FUNCTION_BLOCK Recipe_10018_TripleCookiemitTopping
VAR_INPUT
	execute	: BOOL;
	Order	: DUT_RECIPEORDER;
END_VAR
VAR_OUTPUT
	RecipeInfo	: DUT_RECIPEOFFER;
	RecipeDone	: BOOL;	
	InitDone	: BOOL;
END_VAR
VAR
	StepDone	: BOOL;
	Layercnt	: INT := 0;
	OrderLayers	: INT := 2;
	i : INT;
END_VAR

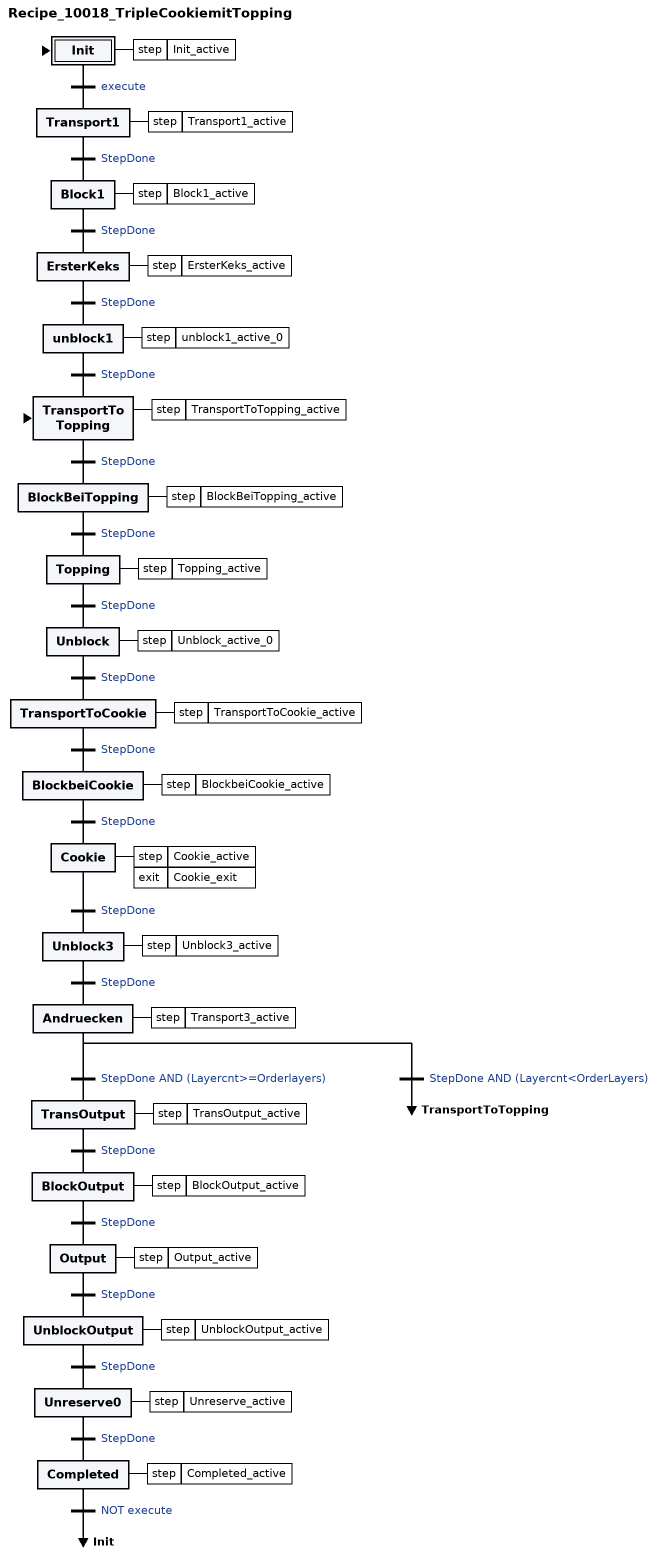
INITIAL_STEP Init:
    Init_active(N);  // step action
END_STEP
TRANSITION FROM Init TO Transport1
    := execute;
END_TRANSITION
STEP Transport1:
    Transport1_active(N);  // step action
END_STEP
TRANSITION FROM Transport1 TO Block1
    := StepDone;
END_TRANSITION
STEP Block1:
    Block1_active(N);  // step action
END_STEP
TRANSITION FROM Block1 TO ErsterKeks
    := StepDone;
END_TRANSITION
STEP ErsterKeks:
    ErsterKeks_active(N);  // step action
END_STEP
TRANSITION FROM ErsterKeks TO unblock1
    := StepDone;
END_TRANSITION
STEP unblock1:
    unblock1_active_0(N);  // step action
END_STEP
TRANSITION FROM unblock1 TO TransportToTopping
    := StepDone;
END_TRANSITION
STEP TransportToTopping:
    TransportToTopping_active(N);  // step action
END_STEP
TRANSITION FROM TransportToTopping TO BlockBeiTopping
    := StepDone;
END_TRANSITION
STEP BlockBeiTopping:
    BlockBeiTopping_active(N);  // step action
END_STEP
TRANSITION FROM BlockBeiTopping TO Topping
    := StepDone;
END_TRANSITION
STEP Topping:
    Topping_active(N);  // step action
END_STEP
TRANSITION FROM Topping TO Unblock
    := StepDone;
END_TRANSITION
STEP Unblock:
    Unblock_active_0(N);  // step action
END_STEP
TRANSITION FROM Unblock TO TransportToCookie
    := StepDone;
END_TRANSITION
STEP TransportToCookie:
    TransportToCookie_active(N);  // step action
END_STEP
TRANSITION FROM TransportToCookie TO BlockbeiCookie
    := StepDone;
END_TRANSITION
STEP BlockbeiCookie:
    BlockbeiCookie_active(N);  // step action
END_STEP
TRANSITION FROM BlockbeiCookie TO Cookie
    := StepDone;
END_TRANSITION
STEP Cookie:
    Cookie_active(N);  // step action
    Cookie_exit(P0);  // exit action
END_STEP
TRANSITION FROM Cookie TO Unblock3
    := StepDone;
END_TRANSITION
STEP Unblock3:
    Unblock3_active(N);  // step action
END_STEP
TRANSITION FROM Unblock3 TO Andruecken
    := StepDone;
END_TRANSITION
STEP Andruecken:
    Transport3_active(N);  // step action
END_STEP
TRANSITION FROM Andruecken TO TransOutput
    := StepDone AND (Layercnt>=Orderlayers);
END_TRANSITION
STEP TransOutput:
    TransOutput_active(N);  // step action
END_STEP
TRANSITION FROM TransOutput TO BlockOutput
    := StepDone;
END_TRANSITION
STEP BlockOutput:
    BlockOutput_active(N);  // step action
END_STEP
TRANSITION FROM BlockOutput TO Output
    := StepDone;
END_TRANSITION
STEP Output:
    Output_active(N);  // step action
END_STEP
TRANSITION FROM Output TO UnblockOutput
    := StepDone;
END_TRANSITION
STEP UnblockOutput:
    UnblockOutput_active(N);  // step action
END_STEP
TRANSITION FROM UnblockOutput TO Unreserve0
    := StepDone;
END_TRANSITION
TRANSITION FROM Andruecken TO TransportToTopping
    := StepDone AND (Layercnt<OrderLayers);
END_TRANSITION
STEP Unreserve0:
    Unreserve_active(N);  // step action
END_STEP
TRANSITION FROM Unreserve0 TO Completed
    := StepDone;
END_TRANSITION
STEP Completed:
    Completed_active(N);  // step action
END_STEP
TRANSITION FROM Completed TO Init
    := NOT execute;
END_TRANSITION

ACTION BlockOutput_active:
StepDone := FALSE;

//Skill auswählen



ExecuteSkill.SkillID 		:= 1315;
ExecuteSkill.SkillName	 	:= 'Block';

ExecuteSkill();

StepDone := ExecuteSkill.Done;
END_ACTION

ACTION Production2_active:
StepDone := FALSE;
RecipeDone := FALSE;
//Skill auswählen
ExecuteSkill.SkillID 		:= 1339;
ExecuteSkill.SkillName	 	:= 'ParameterTESTSKILL1339';


ExecuteSkill.Parameter[0].ID := 10;
ExecuteSkill.Parameter[0].Name := 'Blinkfrequenz';
ExecuteSkill.Parameter[0].Value := Order.UserParameter[0].Value*2;


ExecuteSkill();

StepDone := ExecuteSkill.Done;
END_ACTION

ACTION TransportToCookie_active:
StepDone := FALSE;

//Skill auswählen
ExecuteSkill.SkillID 		:= 1320;
ExecuteSkill.SkillName	 	:= 'Transport';

//Parameter setzen

ExecuteSkill.Parameter[3].ID := 3;
ExecuteSkill.Parameter[3].Name := 'Velocity';
ExecuteSkill.Parameter[3].Value := 400;



ExecuteSkill.Parameter[1].ID :=  1;
ExecuteSkill.Parameter[1].Name := 'TargetPosition X';
ExecuteSkill.Parameter[1].Value := 30 ;
ExecuteSkill.Parameter[1].StringValue := '#DP#2#XPosition';



ExecuteSkill.Parameter[2].ID := 2;
ExecuteSkill.Parameter[2].Name := 'TargetPosition Z';
ExecuteSkill.Parameter[2].Value := ZCookieModule + ZCookieModuleCalibration - ((Layercnt +1) * ( toppingthickness - cookiethickness)) ;

ExecuteSkill();

StepDone := ExecuteSkill.Done;
END_ACTION

ACTION Topping_active:
StepDone := FALSE;

//Skill auswählen
CASE REAL_TO_INT (order.UserParameter[2*LayerCnt].Value) OF
	1: 
		ExecuteSkill.SkillID 		:=  1230;
		ExecuteSkill.SkillName	 	:= 'Strawberry Topping';
	2: 
		ExecuteSkill.SkillID 		:=  1240;
		ExecuteSkill.SkillName	 	:= 'Apple Topping';
	ELSE
		ExecuteSkill.SkillID 		:=  1230;
		ExecuteSkill.SkillName	 	:= 'Strawberry Topping';
END_CASE


//Parameter setzen

ExecuteSkill.Parameter[0].ID := 1;
ExecuteSkill.Parameter[0].Name := 'Amount';
ExecuteSkill.Parameter[0].Value := order.UserParameter[2*LayerCnt + 1].Value ;


(*
ExecuteSkill.Parameter[1].ID := 1;
ExecuteSkill.Parameter[1].Name := 'TaskID';
ExecuteSkill.Parameter[1].Value := 130;
*)
(*
ExecuteSkill.Parameter[2].ID := ;
ExecuteSkill.Parameter[2].Name := '';
ExecuteSkill.Parameter[2].Value := ;
*)

(*
ExecuteSkill.Parameter[3].ID := ;
ExecuteSkill.Parameter[3].Name := '';
ExecuteSkill.Parameter[3].Value := ;
*)

(*
ExecuteSkill.Parameter[4].ID := ;
ExecuteSkill.Parameter[4].Name := '';
ExecuteSkill.Parameter[4].Value := ;
*)

(*
ExecuteSkill.Parameter[5].ID := ;
ExecuteSkill.Parameter[5].Name := '';
ExecuteSkill.Parameter[5].Value := ;
*)

ExecuteSkill();

StepDone := ExecuteSkill.Done;
END_ACTION

ACTION BlockbeiCookie_active:
StepDone := FALSE;

//Skill auswählen
ExecuteSkill.SkillID 		:= 1315;
ExecuteSkill.SkillName	 	:= 'Block';

//Parameter setzen

ExecuteSkill.Parameter[1].ID := 1;
ExecuteSkill.Parameter[1].Name := 'TaskID';
ExecuteSkill.Parameter[1].Value := 130;


(*
ExecuteSkill.Parameter[2].ID := ;
ExecuteSkill.Parameter[2].Name := '';
ExecuteSkill.Parameter[2].Value := ;
*)

(*
ExecuteSkill.Parameter[3].ID := ;
ExecuteSkill.Parameter[3].Name := '';
ExecuteSkill.Parameter[3].Value := ;
*)

(*
ExecuteSkill.Parameter[4].ID := ;
ExecuteSkill.Parameter[4].Name := '';
ExecuteSkill.Parameter[4].Value := ;
*)

(*
ExecuteSkill.Parameter[5].ID := ;
ExecuteSkill.Parameter[5].Name := '';
ExecuteSkill.Parameter[5].Value := ;
*)



ExecuteSkill();

StepDone := ExecuteSkill.Done;
END_ACTION

ACTION Unblock1_active:
StepDone := FALSE;

//Skill auswählen

CASE LREAL_TO_INT (order.UserParameter[2].Value) OF

1:
ExecuteSkill.SkillID 		:= 1316;
ExecuteSkill.SkillName	 	:= 'Unblock';

ExecuteSkill();

StepDone := ExecuteSkill.Done;
ELSE StepDone := TRUE;

END_CASE
END_ACTION

ACTION Transport_active:
StepDone := FALSE;

//Skill auswählen

CASE LREAL_TO_INT (order.UserParameter[2].Value) OF

1:
//Skill auswählen
ExecuteSkill.SkillID 		:= 1320;
ExecuteSkill.SkillName	 	:= 'Transport';

//Parameter setzen

ExecuteSkill.Parameter[3].ID :=3 ;
ExecuteSkill.Parameter[3].Name := 'Velocity';
ExecuteSkill.Parameter[3].Value := 1500;



ExecuteSkill.Parameter[1].ID :=1 ;
ExecuteSkill.Parameter[1].Name := 'TargetPosition X';
ExecuteSkill.Parameter[1].StringValue := '#DP#2#XPosition';
ExecuteSkill.Parameter[1].Value := 200 ;


ExecuteSkill.Parameter[2].ID := 2 ;
ExecuteSkill.Parameter[2].Name := 'TargetPosition Z';
ExecuteSkill.Parameter[2].Value := 90 ;



ExecuteSkill.Parameter[4].ID := 4 ;
ExecuteSkill.Parameter[4].Name := 'Acceleration';
ExecuteSkill.Parameter[4].Value := 4500;


(*
ExecuteSkill.Parameter[5].ID := ;
ExecuteSkill.Parameter[5].Name := '';
ExecuteSkill.Parameter[5].Value := ;
*)



ExecuteSkill();

StepDone := ExecuteSkill.Done;
ELSE StepDone := TRUE;

END_CASE
END_ACTION

ACTION Transport2_active:
StepDone := FALSE;

//Skill auswählen
ExecuteSkill.SkillID 		:= 1320;
ExecuteSkill.SkillName	 	:= 'Transport';

//Parameter setzen

ExecuteSkill.Parameter[3].ID := 3;
ExecuteSkill.Parameter[3].Name := 'Velocity';
ExecuteSkill.Parameter[3].Value := 2800;



ExecuteSkill.Parameter[1].ID :=  1;
ExecuteSkill.Parameter[1].Name := 'TargetPosition X';
ExecuteSkill.Parameter[1].Value := 30 ;
ExecuteSkill.Parameter[1].StringValue := '#DP#2#XPosition';



ExecuteSkill.Parameter[2].ID := 2;
ExecuteSkill.Parameter[2].Name := 'TargetPosition Z';
ExecuteSkill.Parameter[2].Value := 0 ;



ExecuteSkill.Parameter[4].ID := 4;
ExecuteSkill.Parameter[4].Name := 'Acceleration';
ExecuteSkill.Parameter[4].Value := 2000 ;


(*
ExecuteSkill.Parameter[5].ID := ;
ExecuteSkill.Parameter[5].Name := '';
ExecuteSkill.Parameter[5].Value := ;
*)



ExecuteSkill();

StepDone := ExecuteSkill.Done;
END_ACTION

ACTION Block2_active:
StepDone := FALSE;

//Skill auswählen
ExecuteSkill.SkillID 		:= 1315;
ExecuteSkill.SkillName	 	:= 'Block';

//Parameter setzen

ExecuteSkill.Parameter[1].ID := 1;
ExecuteSkill.Parameter[1].Name := 'TaskID';
ExecuteSkill.Parameter[1].Value := 130;


(*
ExecuteSkill.Parameter[2].ID := ;
ExecuteSkill.Parameter[2].Name := '';
ExecuteSkill.Parameter[2].Value := ;
*)

(*
ExecuteSkill.Parameter[3].ID := ;
ExecuteSkill.Parameter[3].Name := '';
ExecuteSkill.Parameter[3].Value := ;
*)

(*
ExecuteSkill.Parameter[4].ID := ;
ExecuteSkill.Parameter[4].Name := '';
ExecuteSkill.Parameter[4].Value := ;
*)

(*
ExecuteSkill.Parameter[5].ID := ;
ExecuteSkill.Parameter[5].Name := '';
ExecuteSkill.Parameter[5].Value := ;
*)



ExecuteSkill();

StepDone := ExecuteSkill.Done;
END_ACTION

ACTION Reserve_active:
StepDone := FALSE;
RecipeDone := FALSE;
//Skill auswählen
ExecuteSkill.SkillID 		:= 1310;
ExecuteSkill.SkillName	 	:= 'Reserve';

//Parameter setzen

ExecuteSkill.Parameter[1].ID := 1;
ExecuteSkill.Parameter[1].Name := 'TaskID';
ExecuteSkill.Parameter[1].Value := 123;


(*
ExecuteSkill.Parameter[2].ID := ;
ExecuteSkill.Parameter[2].Name := '';
ExecuteSkill.Parameter[2].Value := ;
*)

(*
ExecuteSkill.Parameter[3].ID := ;
ExecuteSkill.Parameter[3].Name := '';
ExecuteSkill.Parameter[3].Value := ;
*)

(*
ExecuteSkill.Parameter[4].ID := ;
ExecuteSkill.Parameter[4].Name := '';
ExecuteSkill.Parameter[4].Value := ;
*)

(*
ExecuteSkill.Parameter[5].ID := ;
ExecuteSkill.Parameter[5].Name := '';
ExecuteSkill.Parameter[5].Value := ;
*)



ExecuteSkill();

StepDone := ExecuteSkill.Done;
END_ACTION

ACTION Unblock_active:
StepDone := FALSE;

//Skill auswählen
ExecuteSkill.SkillID 		:= 1316;
ExecuteSkill.SkillName	 	:= 'Unblock';

//Parameter setzen

ExecuteSkill.Parameter[1].ID := 1;
ExecuteSkill.Parameter[1].Name := 'TaskID';
ExecuteSkill.Parameter[1].Value := 125;


(*
ExecuteSkill.Parameter[2].ID := ;
ExecuteSkill.Parameter[2].Name := '';
ExecuteSkill.Parameter[2].Value := ;
*)

(*
ExecuteSkill.Parameter[3].ID := ;
ExecuteSkill.Parameter[3].Name := '';
ExecuteSkill.Parameter[3].Value := ;
*)

(*
ExecuteSkill.Parameter[4].ID := ;
ExecuteSkill.Parameter[4].Name := '';
ExecuteSkill.Parameter[4].Value := ;
*)

(*
ExecuteSkill.Parameter[5].ID := ;
ExecuteSkill.Parameter[5].Name := '';
ExecuteSkill.Parameter[5].Value := ;
*)



ExecuteSkill();

StepDone := ExecuteSkill.Done;
END_ACTION

ACTION Cookie_active:
StepDone := FALSE;
RecipeDone := FALSE;
//Skill auswählen
ExecuteSkill.SkillID 		:= 1010;
ExecuteSkill.SkillName	 	:= 'Cookie ausgeben';





ExecuteSkill();

StepDone := ExecuteSkill.Done;
END_ACTION

ACTION TransOutput_active:
StepDone := FALSE;

//Skill auswählen
ExecuteSkill.SkillID 		:= 1320;
ExecuteSkill.SkillName	 	:= 'Name';

//Parameter setzen

ExecuteSkill.Parameter[3].ID := 3;
ExecuteSkill.Parameter[3].Name := 'Velocity';
ExecuteSkill.Parameter[3].Value := 1500;



ExecuteSkill.Parameter[4].ID := 4 ;
ExecuteSkill.Parameter[4].Name := 'Acceleration';
ExecuteSkill.Parameter[4].Value := 1000 ;



ExecuteSkill.Parameter[1].ID := 1;
ExecuteSkill.Parameter[1].Name := 'TargetPosition X';
ExecuteSkill.Parameter[1].Value := 3200 ;
ExecuteSkill.Parameter[1].StringValue := '#DP#2#XPosition' ;




ExecuteSkill.Parameter[2].ID := 2;
ExecuteSkill.Parameter[2].Name := 'TargetPosition Z';
ExecuteSkill.Parameter[2].Value := ZInputOutput;


(*
ExecuteSkill.Parameter[5].ID := ;
ExecuteSkill.Parameter[5].Name := '';
ExecuteSkill.Parameter[5].Value := ;
*)



ExecuteSkill();

StepDone := ExecuteSkill.Done;
END_ACTION

ACTION TransportToTopping_active:
StepDone := FALSE;

//Skill auswählen
ExecuteSkill.SkillID 		:= 1320;
ExecuteSkill.SkillName	 	:= 'Transport';

//Parameter setzen

ExecuteSkill.Parameter[3].ID := 3;
ExecuteSkill.Parameter[3].Name := 'Velocity';
ExecuteSkill.Parameter[3].Value := 1000;



ExecuteSkill.Parameter[1].ID :=  1;
ExecuteSkill.Parameter[1].Name := 'TargetPosition X';
ExecuteSkill.Parameter[1].Value := 30 ;
ExecuteSkill.Parameter[1].StringValue := '#DP#2#XPosition';



ExecuteSkill.Parameter[2].ID := 2;
ExecuteSkill.Parameter[2].Name := 'TargetPosition Z';
ExecuteSkill.Parameter[2].Value := ZCremeModule + ZCremeModuleCalibration - Layercnt * ( cookiethickness + toppingthickness);

ExecuteSkill();

StepDone := ExecuteSkill.Done;
END_ACTION

ACTION Unblock_active_0:
StepDone := FALSE;

//Skill auswählen
ExecuteSkill.SkillID 		:= 1316;
ExecuteSkill.SkillName	 	:= 'Unblock';

//Parameter setzen

ExecuteSkill.Parameter[1].ID := 1;
ExecuteSkill.Parameter[1].Name := 'TaskID';
ExecuteSkill.Parameter[1].Value := 128 ;


(*
ExecuteSkill.Parameter[2].ID := ;
ExecuteSkill.Parameter[2].Name := '';
ExecuteSkill.Parameter[2].Value := ;
*)

(*
ExecuteSkill.Parameter[3].ID := ;
ExecuteSkill.Parameter[3].Name := '';
ExecuteSkill.Parameter[3].Value := ;
*)

(*
ExecuteSkill.Parameter[4].ID := ;
ExecuteSkill.Parameter[4].Name := '';
ExecuteSkill.Parameter[4].Value := ;
*)

(*
ExecuteSkill.Parameter[5].ID := ;
ExecuteSkill.Parameter[5].Name := '';
ExecuteSkill.Parameter[5].Value := ;
*)



ExecuteSkill();

StepDone := ExecuteSkill.Done;
END_ACTION

ACTION Cookie_exit:
Layercnt := Layercnt +1;
END_ACTION

ACTION Block0_active:
StepDone := FALSE;

//Skill auswählen

CASE LREAL_TO_INT (order.UserParameter[2].Value) OF

1:
ExecuteSkill.SkillID 		:= 1315;
ExecuteSkill.SkillName	 	:= 'Block';

ExecuteSkill();

StepDone := ExecuteSkill.Done;
ELSE StepDone := TRUE;

END_CASE
END_ACTION

ACTION BlockBeiTopping_active:
StepDone := FALSE;

//Skill auswählen
ExecuteSkill.SkillID 		:= 1315;
ExecuteSkill.SkillName	 	:= 'Block';

//Parameter setzen

ExecuteSkill.Parameter[1].ID := 1;
ExecuteSkill.Parameter[1].Name := 'TaskID';
ExecuteSkill.Parameter[1].Value := 130;


(*
ExecuteSkill.Parameter[2].ID := ;
ExecuteSkill.Parameter[2].Name := '';
ExecuteSkill.Parameter[2].Value := ;
*)

(*
ExecuteSkill.Parameter[3].ID := ;
ExecuteSkill.Parameter[3].Name := '';
ExecuteSkill.Parameter[3].Value := ;
*)

(*
ExecuteSkill.Parameter[4].ID := ;
ExecuteSkill.Parameter[4].Name := '';
ExecuteSkill.Parameter[4].Value := ;
*)

(*
ExecuteSkill.Parameter[5].ID := ;
ExecuteSkill.Parameter[5].Name := '';
ExecuteSkill.Parameter[5].Value := ;
*)



ExecuteSkill();

StepDone := ExecuteSkill.Done;
END_ACTION

ACTION Completed_active:
RecipeDone := TRUE;
StepDone := FALSE;
Layercnt := 0;
END_ACTION

ACTION ErsterKeks_active:
StepDone := FALSE;
RecipeDone := FALSE;
//Skill auswählen
ExecuteSkill.SkillID 		:= 1010;
ExecuteSkill.SkillName	 	:= 'Seperate Cookie';


ExecuteSkill();

StepDone := ExecuteSkill.Done;
END_ACTION

ACTION Output_active:
StepDone := FALSE;

//Skill auswählen
ExecuteSkill.SkillID 		:= 1403;
ExecuteSkill.SkillName	 	:= 'Output';

//Parameter setzen

ExecuteSkill.Parameter[1].ID := 1;
ExecuteSkill.Parameter[1].Name := 'TaskID';
ExecuteSkill.Parameter[1].Value := Order.TaskID;


(*
ExecuteSkill.Parameter[2].ID := ;
ExecuteSkill.Parameter[2].Name := '';
ExecuteSkill.Parameter[2].Value := ;
*)

(*
ExecuteSkill.Parameter[3].ID := ;
ExecuteSkill.Parameter[3].Name := '';
ExecuteSkill.Parameter[3].Value := ;
*)

(*
ExecuteSkill.Parameter[4].ID := ;
ExecuteSkill.Parameter[4].Name := '';
ExecuteSkill.Parameter[4].Value := ;
*)

(*
ExecuteSkill.Parameter[5].ID := ;
ExecuteSkill.Parameter[5].Name := '';
ExecuteSkill.Parameter[5].Value := ;
*)



ExecuteSkill();

StepDone := ExecuteSkill.Done;
END_ACTION

ACTION Block1_active:
StepDone := FALSE;

//Skill auswählen
ExecuteSkill.SkillID 		:= 1315;
ExecuteSkill.SkillName	 	:= 'Block';

//Parameter setzen

ExecuteSkill.Parameter[1].ID := 1;
ExecuteSkill.Parameter[1].Name := 'TaskID';
ExecuteSkill.Parameter[1].Value := 127;


(*
ExecuteSkill.Parameter[2].ID := ;
ExecuteSkill.Parameter[2].Name := '';
ExecuteSkill.Parameter[2].Value := ;
*)

(*
ExecuteSkill.Parameter[3].ID := ;
ExecuteSkill.Parameter[3].Name := '';
ExecuteSkill.Parameter[3].Value := ;
*)

(*
ExecuteSkill.Parameter[4].ID := ;
ExecuteSkill.Parameter[4].Name := '';
ExecuteSkill.Parameter[4].Value := ;
*)

(*
ExecuteSkill.Parameter[5].ID := ;
ExecuteSkill.Parameter[5].Name := '';
ExecuteSkill.Parameter[5].Value := ;
*)



ExecuteSkill();

StepDone := ExecuteSkill.Done;
END_ACTION

ACTION Init_active:
RecipeDone := FALSE;

// Initialisation of Recipe Parameters an name etc
RecipeInfo.Name := 'Triple Cookie';
RecipeInfo.Description := 'Three Butter Cookies framing your choosen Toppings';
RecipeInfo.Dummy := FALSE;
RecipeInfo.RecipeID := 10018;	// 
Initdone := TRUE;
FOR i := 0 TO UserParameterCnt DO
	IF Order.UserParameter[i].Value = 0 THEN
		order.UserParameter[i].Value := RecipeInfo.UserParameter[i].Default;
	END_IF
END_FOR

//Parameter 0:

	RecipeInfo.UserParameter[0].Dummy 		:= FALSE;
	RecipeInfo.UserParameter[0].Default		:= 1;
	RecipeInfo.UserParameter[0].Description	:= 'Choose your first Topping (Top Layer)';
	RecipeInfo.UserParameter[0].MaxValue	:= 2;
	RecipeInfo.UserParameter[0].MinValue	:= 1;
	RecipeInfo.UserParameter[0].Name		:= 'Topping';
	RecipeInfo.UserParameter[0].Unit		:= 'Strawberry, Apple';
	RecipeInfo.UserParameter[0].Step		:= 1;

//Parameter 1:

	RecipeInfo.UserParameter[1].Dummy 		:= FALSE;
	RecipeInfo.UserParameter[1].Default		:= 50;
	RecipeInfo.UserParameter[1].Description	:= 'Amount of the selected Topping';
	RecipeInfo.UserParameter[1].MaxValue	:= 100;
	RecipeInfo.UserParameter[1].MinValue	:= 0;
	RecipeInfo.UserParameter[1].Name		:= 'Amount';
	RecipeInfo.UserParameter[1].Unit		:= '';
	RecipeInfo.UserParameter[1].Step		:= 1;

//Parameter 2:
	RecipeInfo.UserParameter[2].Dummy 		:= FALSE;
	RecipeInfo.UserParameter[2].Default		:= 2;
	RecipeInfo.UserParameter[2].Description	:= 'Choose weather you want to include a simulated module';
	RecipeInfo.UserParameter[2].MaxValue	:= 2;
	RecipeInfo.UserParameter[2].MinValue	:= 1;
	RecipeInfo.UserParameter[2].Name		:= 'Virtual Module';
	RecipeInfo.UserParameter[2].Unit		:= 'enabled, disabled';
	RecipeInfo.UserParameter[2].Step		:= 1;

//Parameter 3:
	RecipeInfo.UserParameter[3].Dummy 		:= FALSE;
	RecipeInfo.UserParameter[3].Default		:= 1;
	RecipeInfo.UserParameter[3].Description	:= 'Amount of the selected Topping';
	RecipeInfo.UserParameter[3].MaxValue	:= 100;
	RecipeInfo.UserParameter[3].MinValue	:= 0;
	RecipeInfo.UserParameter[3].Name		:= 'Amount';
	RecipeInfo.UserParameter[3].Unit		:= '';
	RecipeInfo.UserParameter[3].Step		:= 1;
//Parameter 4:

	RecipeInfo.UserParameter[4].Dummy 		:= FALSE;
	RecipeInfo.UserParameter[4].Default		:= 1;
	RecipeInfo.UserParameter[4].Description	:= 'Choose your third Topping';
	RecipeInfo.UserParameter[4].MaxValue	:= 2;
	RecipeInfo.UserParameter[4].MinValue	:= 1;
	RecipeInfo.UserParameter[4].Name		:= 'Topping';
	RecipeInfo.UserParameter[4].Unit		:= 'Strawberry, Apple';
	RecipeInfo.UserParameter[4].Step		:= 1;
	(*
//Parameter 5:

	RecipeInfo.UserParameter[5].Dummy 		:= FALSE;
	RecipeInfo.UserParameter[5].Default		:= 50;
	RecipeInfo.UserParameter[5].Description	:= 'Amount of the selected Topping';
	RecipeInfo.UserParameter[5].MaxValue	:= 100;
	RecipeInfo.UserParameter[5].MinValue	:= 0;
	RecipeInfo.UserParameter[5].Name		:= 'Amount';
	RecipeInfo.UserParameter[5].Unit		:= '';
	RecipeInfo.UserParameter[5].Step		:= 1;
*)
END_ACTION

ACTION Unblock3_active:
StepDone := FALSE;

//Skill auswählen
ExecuteSkill.SkillID 		:= 1316;
ExecuteSkill.SkillName	 	:= 'Unblock';

//Parameter setzen

ExecuteSkill.Parameter[1].ID := 1;
ExecuteSkill.Parameter[1].Name := 'TaskID';
ExecuteSkill.Parameter[1].Value := 131;


(*
ExecuteSkill.Parameter[2].ID := ;
ExecuteSkill.Parameter[2].Name := '';
ExecuteSkill.Parameter[2].Value := ;
*)

(*
ExecuteSkill.Parameter[3].ID := ;
ExecuteSkill.Parameter[3].Name := '';
ExecuteSkill.Parameter[3].Value := ;
*)

(*
ExecuteSkill.Parameter[4].ID := ;
ExecuteSkill.Parameter[4].Name := '';
ExecuteSkill.Parameter[4].Value := ;
*)

(*
ExecuteSkill.Parameter[5].ID := ;
ExecuteSkill.Parameter[5].Name := '';
ExecuteSkill.Parameter[5].Value := ;
*)



ExecuteSkill();

StepDone := ExecuteSkill.Done;
END_ACTION

ACTION Production0_active:
StepDone := FALSE;
RecipeDone := FALSE; 
//simulation ausgewählt?
CASE LREAL_TO_INT (order.UserParameter[2].Value) OF

1:
ExecuteSkill.SkillID 		:= 1337;
ExecuteSkill.SkillName	 	:= 'Testskill';

ExecuteSkill();

StepDone := ExecuteSkill.Done;
ELSE StepDone := TRUE;

END_CASE
END_ACTION

ACTION UnblockOutput_active:
StepDone := FALSE;

//Skill auswählen
ExecuteSkill.SkillID 		:= 1316;
ExecuteSkill.SkillName	 	:= 'Unblock';

//Parameter setzen



(*
ExecuteSkill.Parameter[2].ID := ;
ExecuteSkill.Parameter[2].Name := '';
ExecuteSkill.Parameter[2].Value := ;
*)

(*
ExecuteSkill.Parameter[3].ID := ;
ExecuteSkill.Parameter[3].Name := '';
ExecuteSkill.Parameter[3].Value := ;
*)

(*
ExecuteSkill.Parameter[4].ID := ;
ExecuteSkill.Parameter[4].Name := '';
ExecuteSkill.Parameter[4].Value := ;
*)

(*
ExecuteSkill.Parameter[5].ID := ;
ExecuteSkill.Parameter[5].Name := '';
ExecuteSkill.Parameter[5].Value := ;
*)



ExecuteSkill();

StepDone := ExecuteSkill.Done;
END_ACTION

ACTION Transport1_active:
StepDone := FALSE;

//Skill auswählen
ExecuteSkill.SkillID 		:= 1320;
ExecuteSkill.SkillName	 	:= 'Transport';

//Parameter setzen

ExecuteSkill.Parameter[3].ID := 3;
ExecuteSkill.Parameter[3].Name := 'Velocity';
ExecuteSkill.Parameter[3].Value := 1500;



ExecuteSkill.Parameter[4].ID := 4 ;
ExecuteSkill.Parameter[4].Name := 'Acceleration';
ExecuteSkill.Parameter[4].Value := 1000 ;



ExecuteSkill.Parameter[1].ID := 1;
ExecuteSkill.Parameter[1].Name := 'TargetPosition X';
ExecuteSkill.Parameter[1].Value := 3200 ;
ExecuteSkill.Parameter[1].StringValue := '#DP#2#XPosition' ;




ExecuteSkill.Parameter[2].ID := 2;
ExecuteSkill.Parameter[2].Name := 'TargetPosition Z';
ExecuteSkill.Parameter[2].Value := ZCookieModule + ZCocktailModuleCalibration;


(*
ExecuteSkill.Parameter[5].ID := ;
ExecuteSkill.Parameter[5].Name := '';
ExecuteSkill.Parameter[5].Value := ;
*)



ExecuteSkill();

StepDone := ExecuteSkill.Done;
END_ACTION

ACTION Unreserve_active:
StepDone := FALSE;

//Skill auswählen
ExecuteSkill.SkillID 		:= 1311;
ExecuteSkill.SkillName	 	:= 'Unreserve';

//Parameter setzen

ExecuteSkill.Parameter[1].ID := 1;
ExecuteSkill.Parameter[1].Name := 'TaskID';
ExecuteSkill.Parameter[1].Value := 131;


(*
ExecuteSkill.Parameter[2].ID := ;
ExecuteSkill.Parameter[2].Name := '';
ExecuteSkill.Parameter[2].Value := ;
*)

(*
ExecuteSkill.Parameter[3].ID := ;
ExecuteSkill.Parameter[3].Name := '';
ExecuteSkill.Parameter[3].Value := ;
*)

(*
ExecuteSkill.Parameter[4].ID := ;
ExecuteSkill.Parameter[4].Name := '';
ExecuteSkill.Parameter[4].Value := ;
*)

(*
ExecuteSkill.Parameter[5].ID := ;
ExecuteSkill.Parameter[5].Name := '';
ExecuteSkill.Parameter[5].Value := ;
*)



ExecuteSkill();

StepDone := ExecuteSkill.Done;
END_ACTION

ACTION Unblock2_active:
StepDone := FALSE;

//Skill auswählen
ExecuteSkill.SkillID 		:= 1316;
ExecuteSkill.SkillName	 	:= 'Unblock';

//Parameter setzen

ExecuteSkill.Parameter[1].ID := 1;
ExecuteSkill.Parameter[1].Name := 'TaskID';
ExecuteSkill.Parameter[1].Value := 131;


(*
ExecuteSkill.Parameter[2].ID := ;
ExecuteSkill.Parameter[2].Name := '';
ExecuteSkill.Parameter[2].Value := ;
*)

(*
ExecuteSkill.Parameter[3].ID := ;
ExecuteSkill.Parameter[3].Name := '';
ExecuteSkill.Parameter[3].Value := ;
*)

(*
ExecuteSkill.Parameter[4].ID := ;
ExecuteSkill.Parameter[4].Name := '';
ExecuteSkill.Parameter[4].Value := ;
*)

(*
ExecuteSkill.Parameter[5].ID := ;
ExecuteSkill.Parameter[5].Name := '';
ExecuteSkill.Parameter[5].Value := ;
*)



ExecuteSkill();

StepDone := ExecuteSkill.Done;
END_ACTION

ACTION unblock1_active_0:
StepDone := FALSE;

//Skill auswählen
ExecuteSkill.SkillID 		:= 1316;
ExecuteSkill.SkillName	 	:= 'Unblock';

//Parameter setzen

ExecuteSkill.Parameter[1].ID := 1;
ExecuteSkill.Parameter[1].Name := 'TaskID';
ExecuteSkill.Parameter[1].Value := 128 ;


(*
ExecuteSkill.Parameter[2].ID := ;
ExecuteSkill.Parameter[2].Name := '';
ExecuteSkill.Parameter[2].Value := ;
*)

(*
ExecuteSkill.Parameter[3].ID := ;
ExecuteSkill.Parameter[3].Name := '';
ExecuteSkill.Parameter[3].Value := ;
*)

(*
ExecuteSkill.Parameter[4].ID := ;
ExecuteSkill.Parameter[4].Name := '';
ExecuteSkill.Parameter[4].Value := ;
*)

(*
ExecuteSkill.Parameter[5].ID := ;
ExecuteSkill.Parameter[5].Name := '';
ExecuteSkill.Parameter[5].Value := ;
*)



ExecuteSkill();

StepDone := ExecuteSkill.Done;
END_ACTION

ACTION Transport3_active:
StepDone := FALSE;

//Skill auswählen
ExecuteSkill.SkillID 		:= 1320;
ExecuteSkill.SkillName	 	:= 'Transport';

//Parameter setzen

ExecuteSkill.Parameter[3].ID := 3;
ExecuteSkill.Parameter[3].Name := 'Velocity';
ExecuteSkill.Parameter[3].Value := 2800;



ExecuteSkill.Parameter[1].ID :=  1;
ExecuteSkill.Parameter[1].Name := 'TargetPosition X';
ExecuteSkill.Parameter[1].Value := 30 ;
ExecuteSkill.Parameter[1].StringValue := '#DP#-2#XPosition';



ExecuteSkill.Parameter[2].ID := 2;
ExecuteSkill.Parameter[2].Name := 'TargetPosition Z';
ExecuteSkill.Parameter[2].Value := 90;// ZCookieModule - ZCookieModuleCalibration - 2* Cookiethickness + toppingthickness+ Preasureheight  ;



ExecuteSkill.Parameter[4].ID := 4;
ExecuteSkill.Parameter[4].Name := 'Acceleration';
ExecuteSkill.Parameter[4].Value := 2000 ;


(*
ExecuteSkill.Parameter[5].ID := ;
ExecuteSkill.Parameter[5].Name := '';
ExecuteSkill.Parameter[5].Value := ;
*)



ExecuteSkill();

StepDone := ExecuteSkill.Done;
END_ACTION

END_FUNCTION_BLOCK

(* stored: Version 1.1.0.1, ProductVersion 3.1.0.25
   POU Recipe_10018_TripleCookiemitTopping: Id {35c293d9-a855-4621-991c-8fe2beba9ca6}
   Action BlockOutput_active: Id {074446d1-89b8-4d20-8427-d08b08451a01}
   Action Production2_active: Id {13fb47f7-1ed2-4213-80f0-7c79adf1d406}
   Action TransportToCookie_active: Id {17af7920-8f39-413e-ad0e-663d0bcc4454}
   Action Topping_active: Id {2cb82c9a-a023-458b-86f8-a51686875beb}
   Action BlockbeiCookie_active: Id {33ebe683-30f4-45d2-a737-c9de8ad1aa17}
   Action Unblock1_active: Id {3a205016-96c4-4631-8085-d6e13121b8ed}
   Action Transport_active: Id {50522275-ebaf-458e-95c2-2c4e8c56eb8e}
   Action Transport2_active: Id {50a2aedc-c802-43cb-8069-b660c83db0f4}
   Action Block2_active: Id {5f134dc2-6747-42f2-b0c2-e045c1e90003}
   Action Reserve_active: Id {5f401bc2-1e6e-409d-af80-4924c0799ca2}
   Action Unblock_active: Id {602a6b69-84f2-4e90-9f84-fbefdc5dd0fa}
   Action Cookie_active: Id {66ff8ad2-3785-4db5-bdda-eb892748b77a}
   Action TransOutput_active: Id {7a0639d5-b63d-4ecb-bebd-89e8bec613ac}
   Action TransportToTopping_active: Id {7dda637c-9d5d-47e2-a754-eb5d2485c0ac}
   Action Unblock_active_0: Id {8259acfb-248b-4f4d-889e-6819359f5eae}
   Action Cookie_exit: Id {8414f803-3f1e-4902-9937-0bb17423d579}
   Action Block0_active: Id {9a481e10-3f45-4685-9b36-28940dc0e9f2}
   Action BlockBeiTopping_active: Id {9bcf96d6-5173-422f-8a34-755bcad63f8c}
   Action Completed_active: Id {a7f9d1db-f2f9-46dc-9f89-ce5a1b9250a2}
   Action ErsterKeks_active: Id {c0c0f74f-cfa5-4177-8167-eebe8c00bb9c}
   Action Output_active: Id {c44f2dc4-d8c1-4dd9-93f1-dfd211d851bb}
   Action Block1_active: Id {cc53c5ed-fcac-42cb-a988-0f40d5ea0262}
   Action Init_active: Id {cec50d66-d047-4d5c-9dbb-824294d3a77b}
   Action Unblock3_active: Id {d6b6be0a-4fd7-4b91-835f-a58f0a6357c0}
   Action Production0_active: Id {d70a3a19-a77a-4546-9077-d46d60ee103b}
   Action UnblockOutput_active: Id {ddd7306d-264e-4b40-a3eb-3aee1e34b78e}
   Action Transport1_active: Id {df402391-900f-4146-b34a-02a43a072fa3}
   Action Unreserve_active: Id {e684a77f-1f80-49de-8522-66ffb44cc0b2}
   Action Unblock2_active: Id {ece4eba8-c27e-443d-ba5e-c99703deae09}
   Action unblock1_active_0: Id {fbe8f36f-0777-445a-a2a4-98d8de31871a}
   Action Transport3_active: Id {ffe80e5a-b7ae-4804-8f13-cc73cef7d0f7} *)
